Omron CX-Programmer project NewProject (CX-Programmer 9.50)

# PLC NewPLC1: CP1E N20

## Global symbols (name address type ; comment)
0.00 BOOL  ; PB ON
0.01 BOOL  ; PB RESET
0.02 BOOL  ; PB EMERGENCY
0.03 BOOL  ; SEN 1
0.04 BOOL  ; SEN 2
0.05 BOOL  ; SEN 3
0.06 BOOL  ; SEN 4
100.00 BOOL  ; MTR 1 CONVEYOR
100.01 BOOL  ; MTR 2 POMPA AIR
100.02 BOOL  ; MTR 3 PEMUTAR BOTOL
100.03 BOOL  ; MTR 4 PENGENCANG TUTUP BOTOL
100.04 BOOL  ; SEL VAL TOWER PENGENCANG TUTUP
100.05 BOOL  ; WATER NOZLE
2.00 BOOL  ; K1
2.01 BOOL  ; K2
T000 BOOL  ; T 1
T001 BOOL  ; T 2
T002 BOOL  ; T 3
T003 BOOL  ; T 4
T004 BOOL  ; T 5
T005 BOOL  ; T 6
T006 BOOL  ; T 7
T007 BOOL  ; T 8

## Program NewProgram1 (cyclic task 0)

### Section Section1

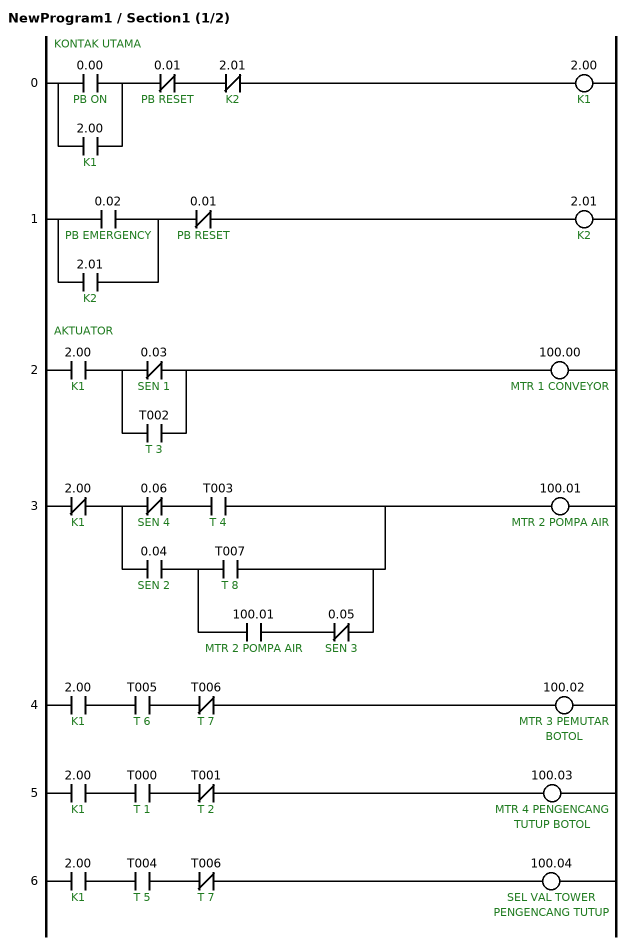
; rung 0: KONTAK UTAMA
LD 0.00  ; PB ON
OR 2.00  ; K1
ANDNOT 0.01  ; PB RESET
ANDNOT 2.01  ; K2
OUT 2.00  ; K1
; rung 1
LD 0.02  ; PB EMERGENCY
OR 2.01  ; K2
ANDNOT 0.01  ; PB RESET
OUT 2.01  ; K2
; rung 2: AKTUATOR
LD 2.00  ; K1
LDNOT 0.03  ; SEN 1
OR T002  ; T 3
ANDLD
OUT 100.00  ; MTR 1 CONVEYOR
; rung 3
LDNOT 2.00  ; K1
LDNOT 0.06  ; SEN 4
AND T003  ; T 4
LD 0.04  ; SEN 2
LD T007  ; T 8
LD 100.01  ; MTR 2 POMPA AIR
ANDNOT 0.05  ; SEN 3
ORLD
ANDLD
ORLD
ANDLD
OUT 100.01  ; MTR 2 POMPA AIR
; rung 4
LD 2.00  ; K1
AND T005  ; T 6
ANDNOT T006  ; T 7
OUT 100.02  ; MTR 3 PEMUTAR BOTOL
; rung 5
LD 2.00  ; K1
AND T000  ; T 1
ANDNOT T001  ; T 2
OUT 100.03  ; MTR 4 PENGENCANG TUTUP BOTOL
; rung 6
LD 2.00  ; K1
AND T004  ; T 5
ANDNOT T006  ; T 7
OUT 100.04  ; SEL VAL TOWER PENGENCANG TUTUP

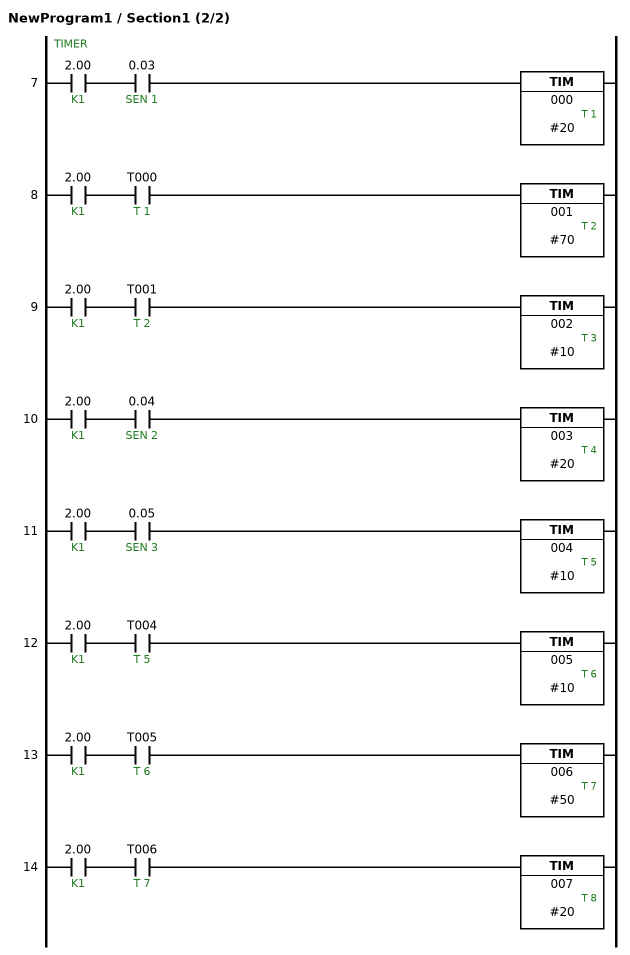
; rung 7: TIMER
LD 2.00  ; K1
AND 0.03  ; SEN 1
TIM 000 #20  ; T 1
; rung 8
LD 2.00  ; K1
AND T000  ; T 1
TIM 001 #70  ; T 2
; rung 9
LD 2.00  ; K1
AND T001  ; T 2
TIM 002 #10  ; T 3
; rung 10
LD 2.00  ; K1
AND 0.04  ; SEN 2
TIM 003 #20  ; T 4
; rung 11
LD 2.00  ; K1
AND 0.05  ; SEN 3
TIM 004 #10  ; T 5
; rung 12
LD 2.00  ; K1
AND T004  ; T 5
TIM 005 #10  ; T 6
; rung 13
LD 2.00  ; K1
AND T005  ; T 6
TIM 006 #50  ; T 7
; rung 14
LD 2.00  ; K1
AND T006  ; T 7
TIM 007 #20  ; T 8

### Section END
; rung 0
END(001)